TYPE ST_InfluxAlarmsInsert :
STRUCT
    {attribute 'TagName' := 'Message'}
	Message		 	: T_MaxString;	// Alarm Message 
    {attribute 'FieldName' := 'ID'}	
	ID			: 	ULINT;
    {attribute 'FieldName' := 'Value'}	
	Value 		: BOOL;
    {attribute 'FieldName' := 'Ack'}	
	Ack			: BOOL;	
END_STRUCT
END_TYPE

(* stored: Version 1.1.0.1, ProductVersion 3.1.4024.6
   DUT ST_InfluxAlarmsInsert: Id {849d499f-7cd8-4623-ab57-0f8c94edb67c} *)
